# EPICS substitutions: jawsApp/Db/jaws_vertical.substitutions
# Create a .db file with records for a set of jaws that consists of vertical blades only (North and South)

file "$(JAWS)/jawsApp/Db/jaws_vertical_header.template" {
    { P=\$(P), JAWS=\$(JAWS), mXN=\$(mXN), mXS=\$(mXS), ASG=\$(ASG=DEFAULT) }
}

file "$(JAWS)/jawsApp/Db/slits.template" {
    { P=\$(P), SLIT=\$(JAWS), M1=\$(mXN), M2=\$(mXS), S1=JN, S2=JS, D1=North, D2=South, GAP=VGAP, DGAP=Vertical, CENTRE=VCENT, DCENTRE=Vertical, ASG=\$(ASG=DEFAULT), EGU=\$(EGU=), CENT_DISP=\$(CENT_DISP=0) }
}
